// TwinCAT 3 PLC project CANSampleCode
// ProgramVersion: 3.1.4023.0
// libraries:
//   Tc2_Standard, * (Beckhoff Automation GmbH)
//   Tc2_System, * (Beckhoff Automation GmbH)
//   Tc3_Module, * (Beckhoff Automation GmbH)
// project tree:
//   DUTs/ ST_TxRxMessage.TcDUT, ST_TxRxQueue.TcDUT
//   / PlcTask.TcTTO
//   POUs/ FB_CANControl.TcPOU, ITF_CANControl.TcIO, MAIN.TcPOU
// real-time tasks:
//   TASK PlcTask: cycle T#10ms, priority 20, ADS port 350

CONFIGURATION CANSampleCode
    RESOURCE PLC ON TwinCAT3
        TASK PlcTask(INTERVAL := T#10ms, PRIORITY := 20);
        PROGRAM MAIN WITH PlcTask : MAIN;
    END_RESOURCE
END_CONFIGURATION

// ---- DUTs/ST_TxRxMessage.TcDUT
{attribute 'pack_mode' := '1'} 
TYPE ST_TxRxMessage :
STRUCT
	dataLength : UINT;
	cobId : UDINT;
	data : ARRAY[0..7] OF BYTE;
END_STRUCT
END_TYPE

// ---- DUTs/ST_TxRxQueue.TcDUT
TYPE ST_TxRxQueue :
STRUCT
	txCounter : UINT;
	rxCounter : UINT;
	noOfMessages : UINT;
	messages : ARRAY[0..9] OF ST_TxRxMessage;
END_STRUCT
END_TYPE

// ---- POUs/ITF_CANControl.TcIO
INTERFACE ITF_CANControl

METHOD M_GetMessage : BOOL
VAR_INPUT
END_VAR
END_METHOD

METHOD M_PushMessage : BOOL
VAR_INPUT
	messageSend : ST_TxRxMessage;
END_VAR
END_METHOD

END_INTERFACE

// ---- POUs/MAIN.TcPOU
PROGRAM MAIN
VAR
END_VAR

END_PROGRAM

// ---- POUs/FB_CANControl.TcPOU
FUNCTION_BLOCK PUBLIC FB_CANControl IMPLEMENTS ITF_CANControl
VAR_INPUT
END_VAR
VAR_OUTPUT
END_VAR
VAR
	rxQueue AT%I* : ST_TxRxQueue;
	txQueue AT%Q* : ST_TxRxQueue;
	i : INT;
	messageRecieved : ST_TxRxMessage;
END_VAR

IF rxQueue.rxCounter <> txQueue.rxCounter THEN
	//if we have recieved a message rxCounter is incremented by interface
	M_GetMessage();
END_IF

METHOD PUBLIC M_GetMessage : BOOL
VAR_INPUT
END_VAR
FOR i := 0 TO rxQueue.noOfMessages DO
	messageRecieved := rxQueue.messages[i];
END_FOR
txQueue.rxCounter := rxQueue.rxCounter;
END_METHOD

METHOD PUBLIC M_PushMessage : BOOL
VAR_INPUT
	messageSend : ST_TxRxMessage;
END_VAR
IF txQueue.txCounter = rxQueue.TxCounter THEN
	FOR i:=0 TO 1 DO
		txQueue.messages[i] := messageSend;
	End_for
	txQueue.noOfMessages := 1;
	txQueue.TxCounter := rxQueue.TxCounter + 1;
END_IF
END_METHOD

END_FUNCTION_BLOCK
